FUNCTION_BLOCK FB_In_Position
VAR_INPUT
	Act_Position	:LREAL;
	Target_Position	:LREAL;	
	Toll_Window		:LREAL;
END_VAR
VAR_OUTPUT
	Axe_In_Pos		:BOOL;

END_VAR
VAR
	_pos_window		:LREAL;
	_neg_window		:LREAL;

END_VAR


_pos_window := Target_Position + Toll_Window;
_neg_window := Target_Position - Toll_Window;

IF (Act_Position >= _neg_window) AND  (Act_Position <= _pos_window) THEN
	Axe_In_Pos := TRUE;
ELSE
	Axe_In_Pos:=FALSE;
END_IF

END_FUNCTION_BLOCK

(* stored: Version 1.1.0.1, ProductVersion 3.1.4022.12
   POU FB_In_Position: Id {6e4e3c5c-8966-4f05-adb8-d562d3f6bed8}, SpecialFunc None *)
